FUNCTION_BLOCK FB_SequenceRND_Calibrate EXTENDS FB_SequenceBase

VAR
	bUseMainPump_A: BOOL := TRUE;  // this boolean is used to keep track of which of the two redudant pumps we should use
END_VAR

VAR_IN_OUT
	devices: ST_RNDDMComponents;
END_VAR

METHOD FB_init : BOOL
VAR_INPUT
	bInitRetains : BOOL; // if TRUE, the retain variables are initialized (warm start / cold start)
	bInCopyCode : BOOL;  // if TRUE, the instance afterwards gets moved into the copy code (online change)
END_VAR
(*
		Here we set the order of things to command, what the commands should be, and also how much time to allow during and between steps
		Every component listed below becomes 'Enabled' at each step
*)

sSequenceName := 'RND-DM Calibrate SEQ';
sSequenceName := 'R&D Dosing Machine Calibrate sequence';
END_METHOD

METHOD populateSteps : ST_SequenceStep
VAR_INPUT

END_VAR
(*
		Here we set the order of things to command, what the commands should be, and also how much time to allow during and between steps
		Every component listed below becomes 'Enabled' at each step
*)

Step1.Device := devices.fbPump_MainPumpA;
Step1.Command := E_DeviceState.RUNNING;
Step1.StepMinDuration := T#5S; 
Step1.DelayUntilNextStep := T#5S;
Step1.WaitForAction := TRUE;
aSequenceSteps[1] :=   Step1;

Step2.Device := devices.fbUVFilter1;
Step2.Command := E_DeviceState.ON;
Step2.StepMinDuration := T#5S;
Step2.DelayUntilNextStep := T#5S;
Step2.WaitForAction := TRUE;
aSequenceSteps[2] :=   Step2;

Step3.Device := devices.fbControlLoop_TankLevel;
Step3.Command := E_DeviceState.ON;
Step3.DelayUntilNextStep := T#5S;
Step3.StepMinDuration := T#5S;
Step3.DelayUntilNextStep := T#5S;
Step3.WaitForAction := TRUE;
aSequenceSteps[3] :=   Step3;

Step4.Device := devices.fbControlLoop_DissOx;
Step4.Command := E_DeviceState.ON;
Step4.DelayUntilNextStep := T#5S;
Step4.StepMinDuration := T#5S;
Step4.DelayUntilNextStep := T#5S;
Step4.WaitForAction := TRUE;
aSequenceSteps[4] :=   Step4;

Step5.Device := devices.fbControlLoop_Dosing;
Step5.Command := E_DeviceState.ON;
Step5.DelayUntilNextStep := T#5S;
Step5.StepMinDuration := T#5S;
Step5.DelayUntilNextStep := T#5S;
Step5.WaitForAction := TRUE;
aSequenceSteps[5] :=   Step5;

Step6.Device := devices.fbValve_Drain;
Step6.Command := E_DeviceState.CLOSED;
Step6.DelayUntilNextStep := T#5S;
Step6.StepMinDuration := T#5S;
Step6.DelayUntilNextStep := T#5S;
Step6.WaitForAction := TRUE;
aSequenceSteps[6] :=   Step6;


nNumberSequenceSteps := 6;  // use this number to limit the number of operations
updateVarIDs();
END_METHOD

END_FUNCTION_BLOCK

(* stored: Version 1.1.0.1, ProductVersion 3.1.4024.12
   POU FB_SequenceRND_Calibrate: Id {7115fecd-f2d3-4eb9-a0a3-4ca3154c0fae}, SpecialFunc None
   Method FB_init: Id {414b4397-5510-4e96-bc8e-fb8069dc395a}
   Method populateSteps: Id {a099bf27-8fc4-4798-84db-f2e047f62806} *)
